(* Logix 5000 project; controller lab_1 vendor 1 type 14 code 96 rev 28.11; software revision 28.00 *)

TASK MainTask (continuous, watchdog 500 ms) : MainProgram

MODULES
   Local : vendor 1 type 14 code 96 (ICP 1, rev 28.11)
      INPUT : vendor 1 type 7 code 2 (ICP 2, rev 3.1, Input RPI 20 ms)
      RELAY_4 : 1756-OW16I (ICP 4, rev 3.1, Output RPI 20 ms)
      Relay_1 : 1756-OW16I (ICP 0, rev 3.3, Output RPI 20 ms)
      Relay_8 : 1756-IF6I (ICP 6, rev 1.1, Input RPI 100 ms)
      Relay_7 : vendor 1 type 10 code 4 (ICP 5, rev 1.12, Output RPI 25 ms)
END_MODULES

PROGRAM MainProgram   (* main routine MainRoutine *)
VAR
   ESTOP : ALIAS FOR Local:2:I.Data.8;
   RED_LIGHT : ALIAS FOR Local:2:I.Data.2;
   run : BOOL;
   RUN_CMD : DINT;
   START : ALIAS FOR Local:2:I.Data.0;
   STOP_PB : ALIAS FOR Local:2:I.Data.9;
END_VAR

ROUTINE MainRoutine   (* ladder *)
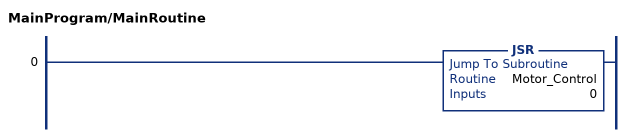
   0: JSR(Motor_Control,0);
END_ROUTINE

ROUTINE Motor_Control   (* ladder *)
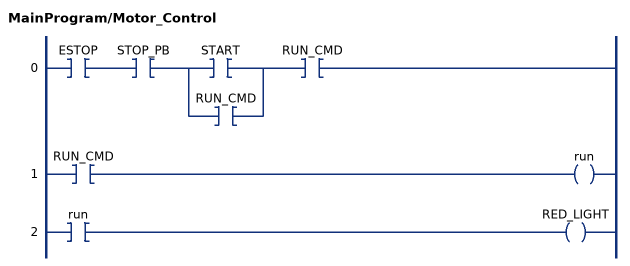
   0: XIC(ESTOP)XIC(STOP_PB)[XIC(START) ,XIC(RUN_CMD) ]XIC(RUN_CMD);
   1: XIC(RUN_CMD)OTE(run);
   2: XIC(run)OTE(RED_LIGHT);
END_ROUTINE
END_PROGRAM
